// TIA Portal V17 export
// export: Created 2021-12-03T08:13:00.860231Z, ExportSetting WithDefaults, DisplayName Totally Integrated Automation Portal, DisplayVersion V17, DisplayName TIA Portal Openness, DisplayVersion V17, DisplayName TIA Portal Version Control Interface, DisplayVersion V17, DisplayName STEP 7 Professional, DisplayVersion V17, DisplayName STEP 7 Safety, DisplayVersion V17, DisplayName WinCC Advanced, DisplayVersion V17
FUNCTION "FC_ScanTransit" : Void   // FC71, FBD
VERSION : 0.1
// stored: AutoNumber false, IsIECCheckEnabled false, UDAEnableTagReadback false
   VAR_TEMP   // added for the SCL form of the ladder/FBD networks
      _w1 : Bool;
   END_VAR
BEGIN

REGION Network 1: Старт
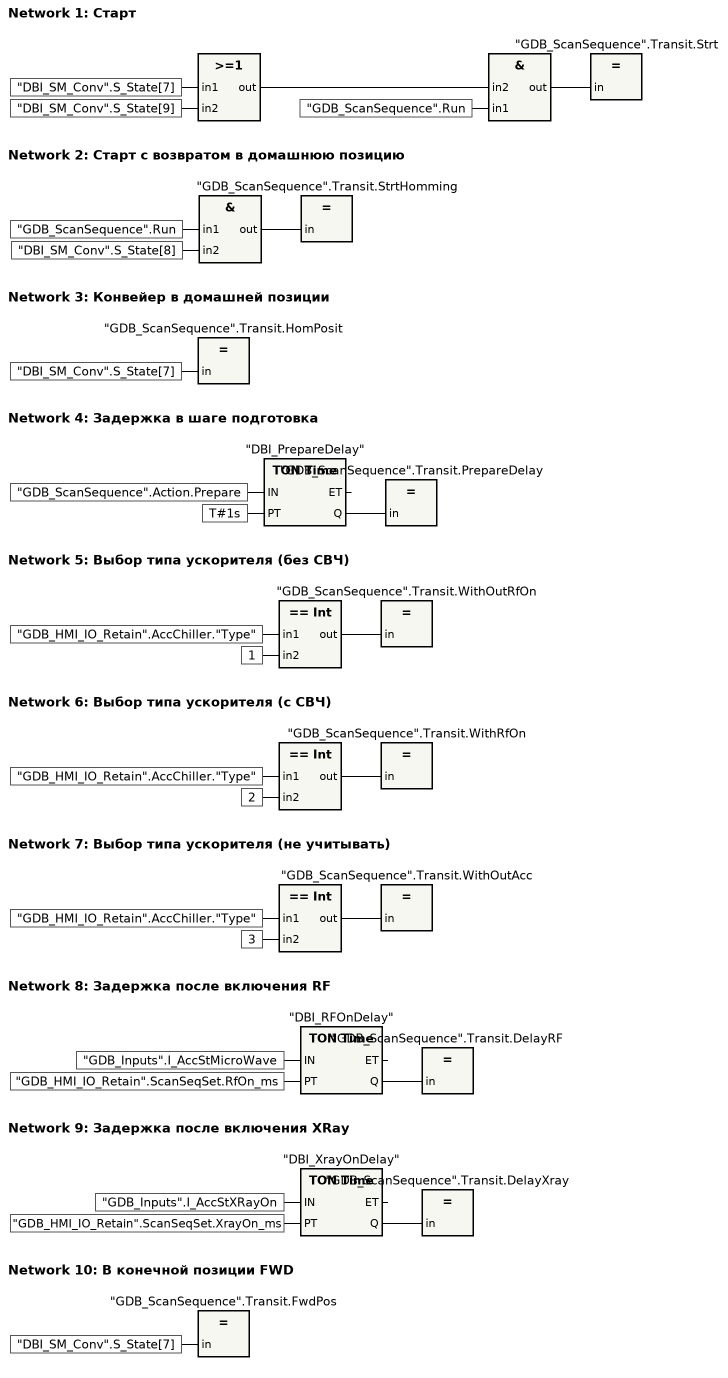
   "GDB_ScanSequence".Transit.Strt := ("DBI_SM_Conv".S_State[7] OR "DBI_SM_Conv".S_State[9]) AND "GDB_ScanSequence".Run;
END_REGION

REGION Network 2: Старт с возвратом в домашнюю позицию
   "GDB_ScanSequence".Transit.StrtHomming := "GDB_ScanSequence".Run AND "DBI_SM_Conv".S_State[8];
END_REGION

REGION Network 3: Конвейер в домашней позиции
   "GDB_ScanSequence".Transit.HomPosit := "DBI_SM_Conv".S_State[7];
END_REGION

REGION Network 4: Задержка в шаге подготовка
   "DBI_PrepareDelay".TON(IN := "GDB_ScanSequence".Action.Prepare, PT := T#1s);
   "GDB_ScanSequence".Transit.PrepareDelay := "DBI_PrepareDelay".Q;
END_REGION

REGION Network 5: Выбор типа ускорителя (без СВЧ)
   "GDB_ScanSequence".Transit.WithOutRfOn := "GDB_HMI_IO_Retain".AccChiller."Type" = 1;
END_REGION

REGION Network 6: Выбор типа ускорителя (с СВЧ)
   "GDB_ScanSequence".Transit.WithRfOn := "GDB_HMI_IO_Retain".AccChiller."Type" = 2;
END_REGION

REGION Network 7: Выбор типа ускорителя (не учитывать)
   "GDB_ScanSequence".Transit.WithOutAcc := "GDB_HMI_IO_Retain".AccChiller."Type" = 3;
END_REGION

REGION Network 8: Задержка после включения RF
   "DBI_RFOnDelay".TON(IN := "GDB_Inputs".I_AccStMicroWave, PT := "GDB_HMI_IO_Retain".ScanSeqSet.RfOn_ms);
   "GDB_ScanSequence".Transit.DelayRF := "DBI_RFOnDelay".Q;
END_REGION

REGION Network 9: Задержка после включения XRay
   "DBI_XrayOnDelay".TON(IN := "GDB_Inputs".I_AccStXRayOn, PT := "GDB_HMI_IO_Retain".ScanSeqSet.XrayOn_ms);
   "GDB_ScanSequence".Transit.DelayXray := "DBI_XrayOnDelay".Q;
END_REGION

REGION Network 10: В конечной позиции FWD
   "GDB_ScanSequence".Transit.FwdPos := "DBI_SM_Conv".S_State[7];
END_REGION

REGION Network 11: В конечной позиции BWD
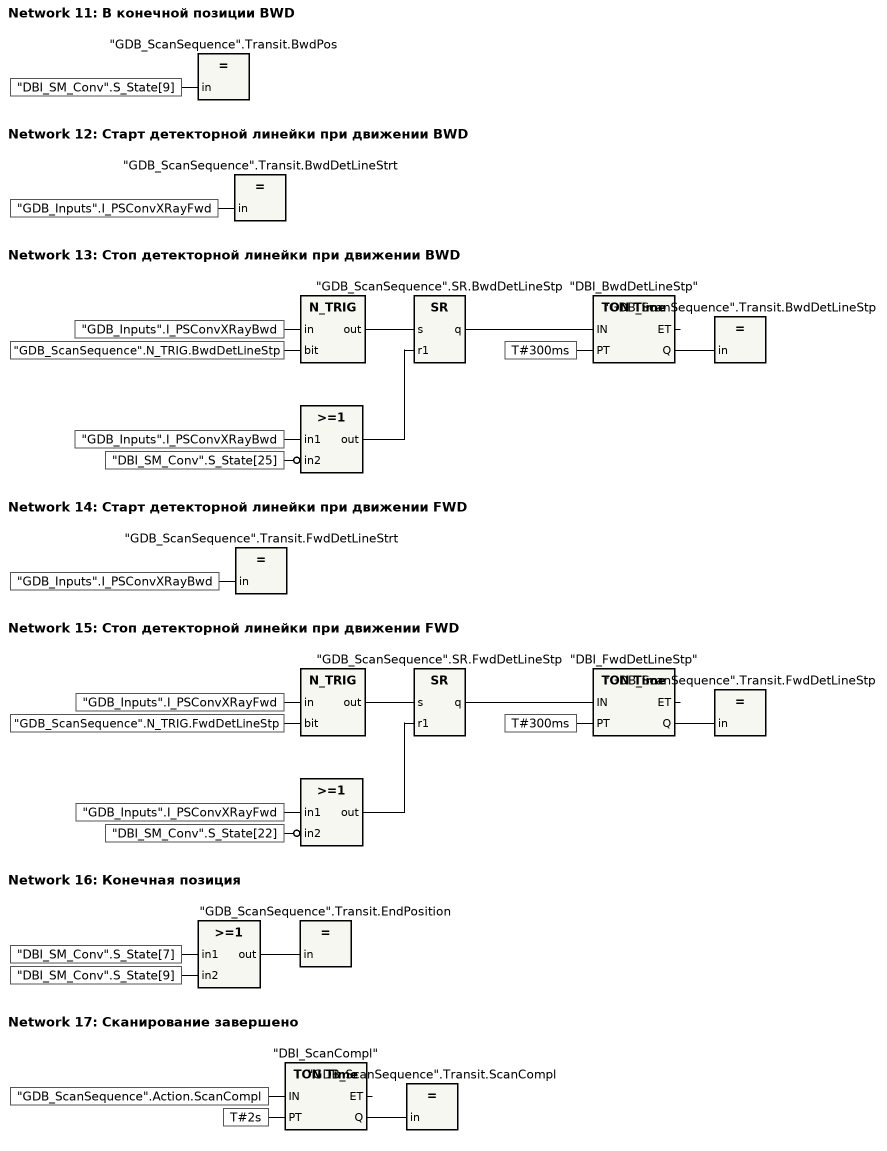
   "GDB_ScanSequence".Transit.BwdPos := "DBI_SM_Conv".S_State[9];
END_REGION

REGION Network 12: Старт детекторной линейки при движении BWD
   "GDB_ScanSequence".Transit.BwdDetLineStrt := "GDB_Inputs".I_PSConvXRayFwd;
END_REGION

REGION Network 13: Стоп детекторной линейки при движении BWD
   #_w1 := NOT "GDB_Inputs".I_PSConvXRayBwd AND "GDB_ScanSequence".N_TRIG.BwdDetLineStp;   // falling edge
   "GDB_ScanSequence".N_TRIG.BwdDetLineStp := "GDB_Inputs".I_PSConvXRayBwd;
   IF #_w1 THEN
       "GDB_ScanSequence".SR.BwdDetLineStp := TRUE;   // SR flip-flop
   END_IF;
   IF "GDB_Inputs".I_PSConvXRayBwd OR NOT "DBI_SM_Conv".S_State[25] THEN
       "GDB_ScanSequence".SR.BwdDetLineStp := FALSE;
   END_IF;
   "DBI_BwdDetLineStp".TON(IN := "GDB_ScanSequence".SR.BwdDetLineStp, PT := T#300ms);
   "GDB_ScanSequence".Transit.BwdDetLineStp := "DBI_BwdDetLineStp".Q;
END_REGION

REGION Network 14: Старт детекторной линейки при движении FWD
   "GDB_ScanSequence".Transit.FwdDetLineStrt := "GDB_Inputs".I_PSConvXRayBwd;
END_REGION

REGION Network 15: Стоп детекторной линейки при движении FWD
   #_w1 := NOT "GDB_Inputs".I_PSConvXRayFwd AND "GDB_ScanSequence".N_TRIG.FwdDetLineStp;   // falling edge
   "GDB_ScanSequence".N_TRIG.FwdDetLineStp := "GDB_Inputs".I_PSConvXRayFwd;
   IF #_w1 THEN
       "GDB_ScanSequence".SR.FwdDetLineStp := TRUE;   // SR flip-flop
   END_IF;
   IF "GDB_Inputs".I_PSConvXRayFwd OR NOT "DBI_SM_Conv".S_State[22] THEN
       "GDB_ScanSequence".SR.FwdDetLineStp := FALSE;
   END_IF;
   "DBI_FwdDetLineStp".TON(IN := "GDB_ScanSequence".SR.FwdDetLineStp, PT := T#300ms);
   "GDB_ScanSequence".Transit.FwdDetLineStp := "DBI_FwdDetLineStp".Q;
END_REGION

REGION Network 16: Конечная позиция
   "GDB_ScanSequence".Transit.EndPosition := "DBI_SM_Conv".S_State[7] OR "DBI_SM_Conv".S_State[9];
END_REGION

REGION Network 17: Сканирование завершено
   "DBI_ScanCompl".TON(IN := "GDB_ScanSequence".Action.ScanCompl, PT := T#2s);
   "GDB_ScanSequence".Transit.ScanCompl := "DBI_ScanCompl".Q;
END_REGION
END_FUNCTION
